Omron CX-Programmer project NewProject (CX-Programmer 9.51)

# PLC NewPLC1: CP1L L

## Global symbols (name address type ; comment)
0.02 BOOL  ; Set F1
0.03 BOOL  ; Set F2
0.04 BOOL  ; Set F3
0.05 BOOL  ; Set F4
100.00 BOOL  ; wy1
100.01 BOOL  ; SMC81_DIR
100.02 BOOL  ; SMC81 driver enable
100.03 BOOL  ; Stepper motor direction
D0 CHANNEL  ; Freq. CLK

## Program NewProgram1 (cyclic task 0)
; SPED function example

### Section Section1

### Section END

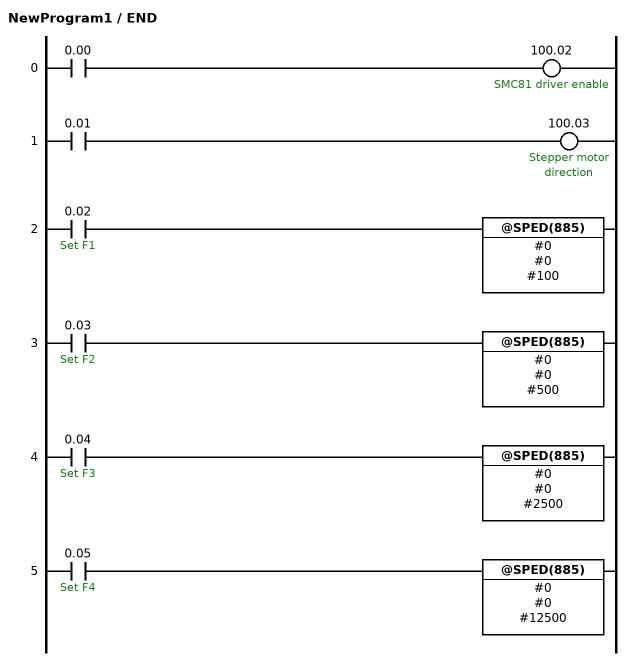
; rung 0
LD 0.00
OUT 100.02  ; SMC81 driver enable
; rung 1
LD 0.01
OUT 100.03  ; Stepper motor direction
; rung 2
LD 0.02  ; Set F1
@SPED(885) #0 #0 #100
; rung 3
LD 0.03  ; Set F2
@SPED(885) #0 #0 #500
; rung 4
LD 0.04  ; Set F3
@SPED(885) #0 #0 #2500
; rung 5
LD 0.05  ; Set F4
@SPED(885) #0 #0 #12500
; rung 6
END(001)